(* IEC 61131-3 sources: PLC-Programming-with-Ladder-Logic-Mini-Project/Solutions/openplc/part6a, 1 file *)

(* ---- part6a.st ---- *)
PROGRAM AutomaticDoorControl
VAR
    Main_Switch : BOOL;
    Object_Detection_Sensor : BOOL;
    Open_Limit_Switch : BOOL;
    Close_Limit_Switch : BOOL;
    Open_Door_Motor : BOOL;
    Close_Door_Motor : BOOL;
    Door_Timer: TON;
    Sequencer: INT;
END_VAR

(* Initial state *)
IF Main_Switch THEN
    IF Sequencer = 0 THEN
        IF Close_Limit_Switch THEN
            Open_Door_Motor := FALSE;
            Close_Door_Motor := FALSE;
            Sequencer := 1;
        END_IF;
    END_IF;

    (* Object detected, open the door *)
    IF Sequencer = 1 THEN
        IF Object_Detection_Sensor AND NOT Open_Limit_Switch THEN
            Open_Door_Motor := TRUE;
            Close_Door_Motor := FALSE;
        ELSIF Open_Limit_Switch THEN
            Open_Door_Motor := FALSE;
            Door_Timer(IN:=TRUE);
            Sequencer := 2;
        END_IF;
    END_IF;

    (* Door is opened for 5 seconds, start closing the door *)
    IF Sequencer = 2 THEN
        IF Door_Timer.Q THEN
            Close_Door_Motor := TRUE;
            Door_Timer(IN:=FALSE);
            Sequencer := 3;
        END_IF;
    END_IF;

    (* Door is fully closed, switch back to initial state *)
    IF Sequencer = 3 THEN
        IF Close_Limit_Switch THEN
            Close_Door_Motor := FALSE;
            Sequencer := 1;
        END_IF;
    END_IF;
END_IF;

END_PROGRAM

CONFIGURATION Config0
    RESOURCE Res0 ON PLC
        TASK task0(INTERVAL := T#20ms, PRIORITY := 0);
        PROGRAM instance0 WITH task0 : AutomaticDoorControl;
    END_RESOURCE
END_CONFIGURATION
